PROGRAM MAIN
VAR
    fbElevator  : FB_Elevator;
END_VAR

// ═══════════════════════════════════════════════════════════════
//  MAIN — Aufzugsteuerung Elevator
//  Aufgerufen von PlcTask alle 10ms
// ═══════════════════════════════════════════════════════════════

fbElevator(
    bEnable := TRUE     // Dauerbetrieb — Not-Halt kommt über GVL_Elevator.bEmergency
);

END_PROGRAM

(* stored: Version 1.1.0.1
   POU MAIN: Id {cfd090f0-c0b3-4ece-b4e6-95adceb6c6bc} *)
